INTERFACE I_Base

METHOD M_Test1 : INT
VAR_INPUT
END_VAR
END_METHOD

PROPERTY P_TestFor : BOOL
GET
END_GET
SET
END_SET
END_PROPERTY

END_INTERFACE

(* stored: Version 1.1.0.1
   Itf I_Base: Id {52fbea3b-879f-4e10-a6a4-a30cd289633e}
   Method M_Test1: Id {e59f5b98-3356-47d7-bdc1-cc4ffebd12c7}
   Property P_TestFor: Id {ea44b91c-f021-4e72-94a8-95bc6f38a944}
   Get Get: Id {69677ebb-9b9d-42a5-99c3-1695f77b0bce}
   Set Set: Id {6e7b6346-5d35-42f5-83fc-2390face48db} *)
